# EPICS IOC start-up script: acalcout/start.iocsh
require calc, 3.7.3
dbLoadRecords("xaxis.db")
dbLoadRecords("ramp.db")
dbLoadRecords("cp_array.db")
